PROGRAM MAIN
VAR
	actualState	:		SafeState := SafeState.Init;	

	blueEdgeDetector : 		FB_EdgeDetector;
	yellowEdgeDetector :	FB_EdgeDetector;
	codeArray : 			ARRAY[0..3] OF BOOL;  // Array mit 4 Elementen vom Typ BOOL
	currentIndex :			INT := 0;
	correctIndex :			INT := 0;
	timer :					TON;
END_VAR

VAR CONSTANT
    lightDuration : TIME := T#5S;
END_VAR

blueEdgeDetector(inputValue:=IO.bBlueButton,DoublePressedTime := 10);
yellowEdgeDetector(inputValue:=IO.bYellowButton,DoublePressedTime := 10);


CASE actualState OF
	SafeState.Init:
	IF NOT(blueEdgeDetector.risingEdge = TRUE AND yellowEdgeDetector.risingEdge = TRUE) THEN
		IF blueEdgeDetector.risingEdge = TRUE THEN
			codeArray[currentIndex] := TRUE;
			currentIndex := currentIndex + 1;
		ELSE
			IF yellowEdgeDetector.risingEdge = TRUE THEN
				codeArray[currentIndex] := FALSE;
				currentIndex := currentIndex + 1;
			END_IF
		END_IF
		IF currentIndex >= 4 THEN
			actualState := SafeState.Close;
			currentIndex := 0;
		END_IF
	END_IF
	;
	SafeState.Close:
		timer(IN:= FALSE,PT:=lightDuration);
		IO.bGreenLight := FALSE;
		IO.bRedLight := FALSE;
		actualState := SafeState.CheckDigit;
	;
	SafeState.CheckDigit:
	IF NOT(blueEdgeDetector.risingEdge = TRUE AND yellowEdgeDetector.risingEdge = TRUE) THEN
		IF blueEdgeDetector.risingEdge = TRUE THEN
			IF codeArray[currentIndex] = TRUE THEN
				correctIndex := correctIndex + 1;
			END_IF
			currentIndex := currentIndex + 1;
		ELSE
			IF yellowEdgeDetector.risingEdge = TRUE THEN
				IF codeArray[currentIndex] = FALSE THEN
					correctIndex := correctIndex + 1;
				END_IF
				currentIndex := currentIndex + 1;
			END_IF
		END_IF

		IF currentIndex >= 4 THEN
			currentIndex := 0;
			IF correctIndex >= 4 THEN
				correctIndex:= 0;
				actualState := SafeState.Open;
			ELSE
				correctIndex := 0;
				actualState := SafeState.WrongCode;
			END_IF
		END_IF
	END_IF
	;
	SafeState.Open:
	IO.bGreenLight := TRUE;
	timer(IN:= TRUE,PT:=lightDuration);
	IF timer.Q = TRUE THEN
		actualState := SafeState.Close;
	END_IF
	;
	SafeState.WrongCode:
	IO.bRedLight := TRUE;
	timer(IN:= TRUE,PT:=lightDuration);
	IF timer.Q = TRUE THEN
		actualState := SafeState.Close;
	END_IF
	;
END_CASE

END_PROGRAM

(* stored: Version 1.1.0.1, ProductVersion 3.1.4024.13
   POU MAIN: Id {94b9cd60-5f9e-4278-9b1e-9a64d0edbf45}, SpecialFunc None *)
